{attribute addProperty BoxType "AX8640-0000-0027"}
{attribute addProperty Id "PSM_PSM_StatuswordAT %I*PSM_PSM_Statusword_C154CB391620WcStateAT %I*WcState_98A4DF7520.250InfoDataAT %I*InfoData_0BDED7BF144180"}
{attribute addProperty CRC "3873554542"}
{attribute addProperty SizeInBites "162"}
{attribute addProperty SizeInBytes "20.25"}
TYPE AX8640_BB1A4FDA :
STRUCT
	{attribute addProperty Name "PSM_PSM_Statusword"}
	PSM_PSM_Statusword : PSM_PSM_Statusword_C154CB39;
	{attribute addProperty Name "WcState"}
	WcState : WcState_98A4DF75;
	{attribute addProperty Name "InfoData"}
	InfoData : InfoData_0BDED7BF;
END_STRUCT
END_TYPE

(* stored: Version 1.2.0.0, ProductVersion 3.1.4024.9
   DUT AX8640_BB1A4FDA: Id {2cae46f5-a3a4-45ac-8295-b713564f4ade} *)
